PROGRAM SchedulerSpecialPeriods
VAR
	fbHVACSchedulerSpecialPeriods:FB_HVACSchedulerSpecialPeriods;
	eDataSecurityType:E_HVACDataSecurityType := E_HVACDataSecurityType.eHVACDataSecurityType_Idle;
	bSetDefault:BOOL;
	bEnable:BOOL;
	dtSystemTime:DT;
	bReset:BOOL;
	arrPeriod:ARRAY[1..20] OF ST_HVACPeriod;
	bOutput:BOOL;
	bEdgeOn:BOOL;
	bEdgeOff:BOOL;
	tNextOn:TIME;
	tNextOff:TIME;
	bInvalidParameter:BOOL;
END_VAR

fbHVACSchedulerSpecialPeriods(
	eDataSecurityType:=eDataSecurityType , 
	bSetDefault:=bSetDefault , 
	bEnable:=bEnable , 
	dtSystemTime:=dtSystemTime, 
	bReset:=bReset, 
	arrPeriod:=arrPeriod, 
	bOutput=>bOutput, 
	bEdgeOn=>bEdgeOn, 
	bEdgeOff=>bEdgeOff, 
	tNextOn=>tNextOn, 
	tNextOff=>tNextOff, 
	bInvalidParameter=>bInvalidParameter);

END_PROGRAM

(* stored: Version 1.1.0.1, ProductVersion 3.1.4024.4
   POU SchedulerSpecialPeriods: Id {a8ef4002-70ed-4a1b-98fa-af5413d321aa}, SpecialFunc None *)
